# B&R Automation Studio project perfxxl (part 6)

#### seriell.c
```c
#ifdef _DEFAULT_INCLUDES
	#include <AsDefault.h>
#endif
/**
                             *******************
******************************* C SOURCE FILE *******************************
**                           *******************                           **
**                                                                         **
** project  : LS JET II                                                    **
** filename : SERIELL.C                                                    **
** version  : 1.12                                                         **
** date     : 15.06.2010                                                   **
**                                                                         **
*****************************************************************************
**                                                                         **
** Abstract                                                                **
** ========                                                                **
** Implementation of serial communication with Faulhaber motor units       **
** - cyclic polling of current position                                    **
** - send commands to a specific motors                                    **
** - request data from a specific motor                                    **
**                                                                         **
**                                                                         **
** Copyright (c) 2006, Krause-Biagosch GmbH                                **
** All rights reserved.                                                    **
**                                                                         **
*****************************************************************************
VERSION HISTORY:
----------------
Version     : 1.00
Date        : 05.09.2002
Revised by  : Herbert Aden
Description : Original version.

Version     : 1.10
Date        : 30.09.2002
Revised by  : Herbert Aden
Description : If a timeout occurs, the Position request is repeated up to 5 times

Version     : 1.11
Date        : 17.10.2006
Revised by  : Herbert Aden
Description : - Code review, style improvement
              - only number of received chars is copied from receive-buffer now
              - RequestData is now local to this module

Version     : 1.12
Date        : 15.06.2010
Revised by  : Herbert Aden
Description : - generate errormessages from FaultStatus (overtemp., current limiting,
                under- or overvoltage)

Version     : 1.13
Date        : 26.04.2011
Revised by  : Herbert Aden
Description : - errormessage delayed to make sure the faultmotor is correctly set
                before the message shows up (avoid error: Motor 0 blahblah)

TODO: Error handling, if system calls fail
*/
#define _SERIELL_C_SRC

/****************************************************************************/
/**                                                                        **/
/**                           INCLUDE FILES                                **/
/**                                                                        **/
/****************************************************************************/
#include <bur/plctypes.h>
#include <string.h>
#include <AsString.h>
#include <dvframe.h>
#include <standard.h>
#include <math.h>

#include "glob_var.h"
#include "sys_lib.h"
#include "motorfunc.h"

/****************************************************************************/
/**                                                                        **/
/**                       DEFINITIONS AND MACROS                           **/
/**                                                                        **/
/****************************************************************************/
#define BROADCAST 127	/* also in motorstop.c !! */
#define DATA_RECEIVED	0
#define STATUS_OK	0

/****************************************************************************/
/**                                                                        **/
/**                           GLOBAL VARIABLES                             **/
/**                                                                        **/
/****************************************************************************/
/*@-exportlocal@*/
/* stop lint from complainig, these are used in another task and therefore GLOBAL*/
_GLOBAL	RTCtime_typ		RTCtime;
_GLOBAL	USINT			MotorTemp[MAXMOTORS],MaxMotorTemp[MAXMOTORS];
_GLOBAL	STRING			MotorFaultStatus[MAXMOTORS][5];
_GLOBAL	DINT			MotorCurrent[MAXMOTORS],MaxMotorCurrent[MAXMOTORS];
/*@+exportlocal@*/

/****************************************************************************/
/**                                                                        **/
/**                      TASK-LOCAL VARIABLES                              **/
/**                                                                        **/
/****************************************************************************/
/* NONE */
_LOCAL	BOOL			GetMotorCurrent;			/* command to get the motor current*/
_LOCAL	UINT            FaultMotor;                 /* for Alarmmessage */
_LOCAL	DINT BufLng;
_LOCAL	STRING DebugBuf[64];

/****************************************************************************/
/**                                                                        **/
/**                    MODULE-LOCAL VARIABLES                              **/
/**                                                                        **/
/****************************************************************************/
static	UINT 			Counter;
static	UINT 			SendWaitCounter;
static	UINT			GetTempStep;
static	UINT			GetTempMotor;
static	USINT			lastSecond;
static	UINT			SecondCounter;
static	BOOL			xopenOK;					/* Opening the interface was successful*/
static	INT 			i;
static 	USINT 			RequestData[READDATALENGTH]; 			/* array for requested Data */
static 	char 			StringDevice[30], StringMode[30]; 		/* initialize strings for FRM_xopen */
static 	UINT 			timeout;
static	UINT 			Motor;						/* index variable for polling loop*/
static	BOOL 			StopPolling;				/* stop polling loop to send a command*/
static	UINT 			PollingStep;
static	UINT 			RequestStep;
static 	UINT			ResendCounter;
static	BOOL			GetMotorCurrentMem;			/* to detect changing of command*/
static	INT				Error;						/* Error Number for debugging*/
static	INT				ReceivedChar;
static	char		    tmp[20];
static	FRM_xopen_typ 	FrameXOpenStruct;
static	FRM_close_typ 	FrameCloseStruct;
static	XOPENCONFIG 	XOpenConfigStruct;
static	FRM_gbuf_typ 	FrameGetBufferStruct;
static	FRM_rbuf_typ 	FrameReleaseBufferStruct;
static	FRM_robuf_typ 	FrameReleaseOutputBufferStruct;
static	FRM_write_typ 	FrameWriteStruct;
static 	FRM_read_typ 	FrameReadStruct;
static  TON_10ms_typ    Alarm36Delay,Alarm37Delay,Alarm38Delay,Alarm39Delay;

/****************************************************************************/
/**                                                                        **/
/**                          LOCAL FUNCTIONS                               **/
/**                                                                        **/
/****************************************************************************/

/**
 * Return the next motor-number in the row, skipping those that are not
 * used in differently equipped machines
 *
 * Input Parameter: Current motor-number
 *
 * Returns        : Next motor-number
 *
 */
static UINT	NextMotor(UINT lMotor)
{
	lMotor++;
	if(lMotor == FEEDER_HORIZONTAL && !GlobalParameter.FlexibleFeeder)
		lMotor++;
	if(lMotor == ADJUSTER)
		lMotor++;
	if(lMotor == SHUTTLE)
		lMotor++;
	if(lMotor == DELOADER_TURN && GlobalParameter.DeloaderTurnStation != DELOADER_AND_TURNSTATION)
		lMotor++;
	if(lMotor == DELOADER_HORIZONTAL && GlobalParameter.DeloaderTurnStation == NO_DELOADER)
		lMotor++;

	if(lMotor > MotorsConnected)
		lMotor = 1;

	return lMotor;
}

/**
 * Auxiliary function to handle timeout while reading from serial interface
 *
 * Input Parameter: ----
 *
 * Returns        : ----
 *
 */
static void HandleTimeout(int returnstep)
{
	Error = 5; 						/* set error level for FRM_read */
	timeout++;
	if (timeout == 60) /* 60*cyclic (->300ms) time no answer */
	{
		if(ResendCounter == 5) /*5 times tried? -> error*/
		{
			ResendCounter = 0;
			Motors[Motor].Error = TRUE;
			Motors[Motor].Moving = FALSE;
			Motors[Motor].MovingPlus = FALSE;
			Motors[Motor].MovingMinus = FALSE;
			Motors[Motor].ReferenceOk = FALSE;
			Motor = NextMotor(Motor);
			if(Motor == 1)
				Counter++;

			PollingStep = 0;
		}
		else
		{
			ResendCounter++;
			PollingStep = /*1*/returnstep;
		}
	}
}

/**
 * Auxiliary function to handle error while writing to serial interface
 *
 * Input Parameter: ----
 *
 * Returns        : ----
 *
 */
static void HandleWriteError(void)
{
	/* initialize release output buffer structure */
	FrameReleaseOutputBufferStruct.buffer = FrameGetBufferStruct.buffer;
	FrameReleaseOutputBufferStruct.buflng = FrameGetBufferStruct.buflng;
	FRM_robuf(&FrameReleaseOutputBufferStruct); 	/* release output buffer */

	Error = 3; 					/* set error level for FRM_write */

	if (FrameReleaseOutputBufferStruct.status != 0) 		/* check status */
	{
		Error = 4; 				/* set error level for FRM_robuf */
	}
}

/**
 * Auxiliary function to handle error while writing to serial interface
 *
 * Input Parameter: ----
 *
 * Returns        : ----
 *
 * TODO: Error handling
 */
static void ReleaseBuffer(void)
{
	/* initialize release buffer structure */
	FrameReleaseBufferStruct.buffer = FrameReadStruct.buffer;	/* get adress of read buffer */
	FrameReleaseBufferStruct.buflng = FrameReadStruct.buflng; 	/* get length of read buffer */

	FRM_rbuf(&FrameReleaseBufferStruct); 			/* release read buffer */

	if (FrameReleaseBufferStruct.status != 0) 				/* check status */
	{
		Error = 6; 					/* set error level for FRM_rbuf */
	}
}

/****************************************************************************/
/** Init function, executed once at startup                                **/
/****************************************************************************/
_INIT void InitProgram(void)
{
	Alarm36Delay.IN = FALSE;
	Alarm37Delay.IN = FALSE;
	Alarm38Delay.IN = FALSE;
	Alarm39Delay.IN = FALSE;
	GetMotorCurrent = FALSE;
	GetMotorCurrentMem = FALSE;
	GetTempMotor = 1;
	lastSecond = US(0);
	SecondCounter = 0;
	for(i=0;i<MAXMOTORS;i++)
	{
		MotorTemp[i] = US(0);
		MaxMotorTemp[i] = US(0);
		MotorCurrent[i] = L(0);
		MaxMotorCurrent[i] = L(0);
	}

	/* initialize start values */
	Motor = 1;
/* Motor Nummern sind 1,2,3,6,9
 * um die Zuordnung zwischen Adr. und Fkt. wie beim Jet2 zu haben
 */
	MotorsConnected = 10;
	SendWaitCounter=0;
	Counter = 0;
	StopPolling = FALSE;
	ResendCounter = 0;
	xopenOK = 0;
	strcpy(&StringDevice[0], "IF1"); 							/* interface #1 */
	strcpy(&StringMode[0], "/BD=19200 /PA=N /DB=8 /SB=1"); 		/* RS232 interface, 19200 BAUD, no parity, 8 data bits, 1 stop bit */

	/* initialize config structure */
	XOpenConfigStruct.idle = 6;                           	/* in Zeichenlängen*/
	XOpenConfigStruct.delimc = 1;
	XOpenConfigStruct.delim[0] = (unsigned char)10;				/* LF */
	XOpenConfigStruct.delim[1] = (unsigned char)13;				/* CR */
	XOpenConfigStruct.tx_cnt = 6;
	XOpenConfigStruct.rx_cnt = 6;
	XOpenConfigStruct.tx_len = 64;
	XOpenConfigStruct.rx_len = 64;
	XOpenConfigStruct.argc = 0;
	XOpenConfigStruct.argv = 0;

	/* initialize open structure */
	FrameXOpenStruct.enable = TRUE;
	FrameXOpenStruct.device = (UDINT) StringDevice;
	FrameXOpenStruct.mode = (UDINT) StringMode;
	FrameXOpenStruct.config = (UDINT) &XOpenConfigStruct;

	FRM_xopen(&FrameXOpenStruct); 						/* open an interface */

	if (FrameXOpenStruct.status == 0) 					/* check status */
	{
		xopenOK = TRUE;									/* set error level for FRM_xopen */

		/* initialize get buffer structure */
		FrameGetBufferStruct.enable = TRUE;
		FrameGetBufferStruct.ident = FrameXOpenStruct.ident;				/* get ident */

		/* initialize write structure */
		FrameWriteStruct.enable = TRUE;
		FrameWriteStruct.ident  = FrameXOpenStruct.ident;					/* get ident */

		/* initialize release output buffer structure */
		FrameReleaseOutputBufferStruct.enable = TRUE;
		FrameReleaseOutputBufferStruct.ident = FrameXOpenStruct.ident;		/* get ident */

		/* initialize read structure */
		FrameReadStruct.enable = TRUE;
		FrameReadStruct.ident = FrameXOpenStruct.ident;						/* get ident */

		/* initialize release buffer structure */
		FrameReleaseBufferStruct.enable = TRUE;
		FrameReleaseBufferStruct.ident = FrameXOpenStruct.ident;			/* get ident */

		/* initialize close structure */
		FrameCloseStruct.enable = TRUE;
		FrameCloseStruct.ident = FrameXOpenStruct.ident;					/* get ident */
	}
	else
	{
		xopenOK = FALSE;
	}
}

/****************************************************************************/
/** Cyclic function                                                        **/
/****************************************************************************/
_CYCLIC void CyclicProgram(void)
{
/*HA 24.02.04 V1.76 reset MaxCurrent on activating measurement*/
	if ( GetMotorCurrent && !GetMotorCurrentMem )
		for(i=0;i<MAXMOTORS;i++)
			MaxMotorCurrent[i] = 0;
	GetMotorCurrentMem = GetMotorCurrent;

	if (xopenOK != FALSE)
	{
/******************************************************************/
/* Cyclic polling of current Positions */
/******************************************************************/
		switch (PollingStep)
		{
			case 0:
			{
				if(StopPolling) break;
				/*Safety: priority 0 doesn't make sense*/
				if(Motors[Motor].Parameter.Priority == US(0)) Motors[Motor].Parameter.Priority = US(1);

				if( (Counter % Motors[Motor].Parameter.Priority) == 0  )
				{
					PollingStep = 100;
				}
				else
				{
					Motor = NextMotor(Motor);
					if(Motor == 1)
						Counter++;
				}
				ResendCounter = 0;
				break;
			}

/* clear buffer from any unwanted msg */
			case 100:
			{
				/* initialize read structure */
				FRM_read(&FrameReadStruct); 						/* read data form interface */

				if (FrameReadStruct.status == DATA_RECEIVED) 					/* Data received */
				{
					ReleaseBuffer();
				}
				ResendCounter = 0;
				PollingStep = 1;
				break;
			}

/* 1st Step: send the POS command */
			case 1:
			{
				FRM_gbuf(&FrameGetBufferStruct); 				/* get send buffer */

				if (FrameGetBufferStruct.status == 0) 			/* check status */
				{
					size_t length = 4; /* length of "xPOS" */
					char *ptr = (char *)FrameGetBufferStruct.buffer;
				/*fill the buffer */
					(void) itoa(L(Motor),(UDINT) ptr);
					strcat(ptr,"POS\r\n");
					length = strlen(ptr);

					/* initialize write structure */
					FrameWriteStruct.buffer = FrameGetBufferStruct.buffer;
					FrameWriteStruct.buflng = length+1;
					FRM_write(&FrameWriteStruct); 				/* write data to interface */

					if (FrameWriteStruct.status != 0) 			/* check status */
					{
						HandleWriteError();
					}
				}
	/*TODO: Fehler auswerten wenn getBuffer fehlschlägt (8071)*/
				PollingStep++;
				timeout = 0;
				break;
			}
/* wait for the answer of Motor*/
			case 2:
			{
				/* initialize read structure */
				FRM_read(&FrameReadStruct); 						/* read data form interface */

				if (FrameReadStruct.status == DATA_RECEIVED) 					/* Data received */
				{
					BufLng = FrameReadStruct.buflng;
					strncpy(DebugBuf,((char *)FrameReadStruct.buffer),sizeof(DebugBuf));
					DebugBuf[BufLng] = '\0';
					if( (((char *)FrameReadStruct.buffer)[0] == '-')
					 || (   (((char *)FrameReadStruct.buffer)[0] >= '0')
					      &&(((char *)FrameReadStruct.buffer)[0] <= '9')
					    )
					  )
					{
						Motors[Motor].LastPosition = Motors[Motor].Position;
						Motors[Motor].Position = atoi( FrameReadStruct.buffer);
	/*@-realcompare@*/
						if(Motors[Motor].Parameter.IncrementsPerMm > 1.0)
							Motors[Motor].Position_mm = Motors[Motor].Position / Motors[Motor].Parameter.IncrementsPerMm;
	/*@+realcompare@*/

						if (Motor == ADJUSTER ||  Motor == CONVEYORBELT)
						{
							AbsMotorPos[Motor] = Motors[Motor].Position;
							AbsMotorPosMm[Motor] = Motors[Motor].Position_mm;
						}
						else
						{
							AbsMotorPos[Motor] = abs(Motors[Motor].Position);
							AbsMotorPosMm[Motor] = fabs(Motors[Motor].Position_mm);
						}

						if( labs(Motors[Motor].Position) > labs(Motors[Motor].LastPosition) )
						{
							Motors[Motor].MovingPlus = TRUE;
							Motors[Motor].MovingMinus = FALSE;
						}
						else
						{
							Motors[Motor].MovingPlus = FALSE;
							Motors[Motor].MovingMinus = TRUE;
						}

						if( labs(Motors[Motor].LastPosition - Motors[Motor].Position) > 100)
							Motors[Motor].Moving = TRUE;
						else
						{
							Motors[Motor].Moving = FALSE;
							Motors[Motor].MovingPlus = FALSE;
							Motors[Motor].MovingMinus = FALSE;
						}

						Motors[Motor].Error = FALSE;
					}
					ReleaseBuffer();
					if ( GetMotorCurrent )
					{
						PollingStep++;
						break;
					}
					else
					{
						Motor = NextMotor(Motor);
						if(Motor == 1)
							Counter++;

						PollingStep = 0;
						ResendCounter = 0;
						break;
					}
				}
				else	/* No data received or any error*/
				{
					HandleTimeout(1);
				}
				break;
			}
/* send the "get current" command*/
			case 3:
			{
					FRM_gbuf(&FrameGetBufferStruct); 				/* get send buffer */

					if (FrameGetBufferStruct.status == 0) 			/* check status */
					{
						size_t length = 4;
						char *ptr = (char *)FrameGetBufferStruct.buffer;
				/*fill the buffer */
						(void) itoa(L(Motor),(UDINT) ptr);
						strcat(ptr,"GRC\r\n"); /*actual current (Get Real Current)*/
						length = strlen(ptr);

					/* initialize write structure */
						FrameWriteStruct.buffer = FrameGetBufferStruct.buffer;		/* get adress of send buffer */
						FrameWriteStruct.buflng = length+1;

						FRM_write(&FrameWriteStruct); 				/* write data to interface */

						if (FrameWriteStruct.status != 0) 			/* check status */
						{
							HandleWriteError();
						}
					}
	/*TODO: Fehler auswerten wenn getBuffer fehlschlägt (8071)*/
					PollingStep++;
					timeout = 0;
					break;
			}

/* wait for the answer of Motor on GRC*/
			case 4:
			{
				/* initialize read structure */
				FRM_read(&FrameReadStruct); 						/* read data form interface */

				if (FrameReadStruct.status == DATA_RECEIVED) 					/* Data received */
				{
					if( (((char *)FrameReadStruct.buffer)[0] == '-')
					 || (   (((char *)FrameReadStruct.buffer)[0] >= '0')
					      &&(((char *)FrameReadStruct.buffer)[0] <= '9')
					    )
					  )
					{
						MotorCurrent[Motor] = atoi( FrameReadStruct.buffer);
						if ( MotorCurrent[Motor] > MaxMotorCurrent[Motor] )
							MaxMotorCurrent[Motor] = MotorCurrent[Motor];
					}
					ReleaseBuffer();

					Motor = NextMotor(Motor);
					if(Motor == 1)
						Counter++;

					PollingStep = 0;
					ResendCounter = 0;
					break;
				}
				else	/* No data received or any error*/
				{
					HandleTimeout(3);
				}
				break;
			}

		} /*switch*/

/******************************************************************/
/* requesting of Parameter */
/******************************************************************/
		switch (RequestStep)
		{
			case 0:
			{
				if(SerialCmd.Send == FALSE) break; /*wait for send command*/

				StopPolling = TRUE;
				if(PollingStep == 0)	/*wait for polling to stop*/
					RequestStep++;
				break;
			}
/* 1st Step: send the command */
			case 1:
			{
				FRM_gbuf(&FrameGetBufferStruct); 				/* get send buffer */

				if (FrameGetBufferStruct.status == STATUS_OK)
				{
					size_t length=0; /* length */
					char *ptr = (char *)FrameGetBufferStruct.buffer;
				/*fill the buffer */
					if( SerialCmd.SendMotor != BROADCAST )  /*no BROADCAST, so the address must be first*/
					{
						(void)itoa(L(SerialCmd.SendMotor),(UDINT) ptr);
						strcat(ptr,(char *) SerialCmd.CmdString);
					}
					else
						strcpy(ptr,(char *) SerialCmd.CmdString);

/* build the final commandstring from given parameters*/
					if (SerialCmd.UseParameter)
					{
						if (SerialCmd.UseRefDirection)
						{
				/*
				 * for absolute positioning:
				 * if Reference direction positive then the way to move is in negative direction
				 * therefore labs(SerialCmd.Parameter)
				*/
							if (STREQ(SerialCmd.CmdString,CMD_ABSOLUTE_POS))
							{
								if( (SerialCmd.SendMotor == CONVEYORBELT) || (SerialCmd.SendMotor == ADJUSTER) )
								{
							/*
							 * special case: the belt drives are able to move in a position below 0
							 * so this is allowed here in that special case
							*/
									(void)itoa(SerialCmd.Parameter,(UDINT) &tmp[0]);
								}
								else
								{
									if (Motors[SerialCmd.SendMotor].Parameter.ReferenceDirectionNegative == FALSE)
										strcat(ptr,"-");
									(void)itoa(labs(SerialCmd.Parameter),(UDINT) &tmp[0]);
								}
							}
							else
				/*
				 * for relative positioning:
				 * moving towards reference pos. must be given as negative values
				 * UseRefDirection must be TRUE
				 * the same applies for speed setting (V-command)
				*/

							if ( (STREQ(SerialCmd.CmdString,CMD_RELATIVE_POS))
								||
								(STREQ(SerialCmd.CmdString,CMD_MOVE_AT)))
							{
								if(Motors[SerialCmd.SendMotor].Parameter.ReferenceDirectionNegative)
								{
									if (SerialCmd.Parameter < 0L)
										strcat(ptr,"-");
								}
								else
								{
									if (SerialCmd.Parameter > 0L)
										strcat(ptr,"-");
								}
								(void)itoa(labs(SerialCmd.Parameter),(UDINT) &tmp[0]);
							}
						}
						else /* don't use RefDirection: take Parameter just as it's given */
							(void)itoa(SerialCmd.Parameter,(UDINT) &tmp[0]);

						strcat(ptr,tmp);
					}
					strcat(ptr,"\r\n");
					length = strlen(ptr);

					/* initialize write structure */
					FrameWriteStruct.buffer = FrameGetBufferStruct.buffer;	/* get adress of send buffer */
					FrameWriteStruct.buflng = length+1; 					/* set length of send buffer */

					FRM_write(&FrameWriteStruct); 				/* write data to interface */

					if (FrameWriteStruct.status != 0) 			/* check status */
					{
						HandleWriteError();
					}
				}
				RequestStep++;
				timeout = 0;
				break;
			}
/* wait for the answer of Motor*/
			case 2:
			{
				/* no request: go on*/
				if(SerialCmd.Request == FALSE)
				{
					SendWaitCounter++;
					if(SendWaitCounter > 6)
					{
						SendWaitCounter=0;
						SerialCmd.Request = FALSE;
						SerialCmd.Send = FALSE;
						StopPolling = FALSE;
						RequestStep = 0;
					}
/* HA 13.02.04 V1.76 no request (command only): leave the code immediately */
					break;
				}
/* otherwise go ahead waiting for answer*/

				/* initialize read structure */
				FRM_read(&FrameReadStruct); 						/* read data form interface */

				if (FrameReadStruct.status == DATA_RECEIVED) 					/* Data received */
				{
					ReceivedChar = (INT) FrameReadStruct.buflng;
					memcpy(RequestData, (USINT*)FrameReadStruct.buffer, (size_t)ReceivedChar); /* copy read data into array */
					Motors[SendMotor].Error = FALSE;

					ReleaseBuffer();

					RequestStep = 0;
					SerialCmd.Request = FALSE;
					SerialCmd.Send = FALSE;
					StopPolling = FALSE;
				}
				else	/* No data received or any error*/
				{
					ReceivedChar = 0;
					Error = 5; 						/* set error level for FRM_read */
					timeout++;
					if (timeout == 60) /* 60*cyclic time no answer */
					{
						RequestStep = 0;
						SerialCmd.Request = FALSE;
						SerialCmd.Send = FALSE;
						StopPolling = FALSE;
						Motors[SerialCmd.SendMotor].Error = TRUE;
						Motors[SerialCmd.SendMotor].Moving = FALSE;
						Motors[SerialCmd.SendMotor].MovingPlus = FALSE;
						Motors[SerialCmd.SendMotor].MovingMinus = FALSE;
					}
				}
				break;
			}
		} /*switch*/

	} /*if (xopenOK == 1)*/

/******************************************************************************************************/
/******************************************************************************************************/
/******************************************************************************************************/
/* Alarm 36 bis 39 5s verzögern, damit der Faultmotor auch sicher eingetragen wurde */
	Alarm36Delay.PT = 500;
	TON_10ms(&Alarm36Delay);
	AlarmBitField[36] = Alarm36Delay.Q;

	Alarm37Delay.PT = 500;
	TON_10ms(&Alarm37Delay);
	AlarmBitField[37] = Alarm37Delay.Q;

	Alarm38Delay.PT = 500;
	TON_10ms(&Alarm38Delay);
	AlarmBitField[38] = Alarm38Delay.Q;

	Alarm39Delay.PT = 500;
	TON_10ms(&Alarm39Delay);
	AlarmBitField[39] = Alarm39Delay.Q;

	switch (GetTempStep)
	{
/* get Temperature every 5 seconds*/
		case 0:
		{
			int CurrentMotor=1,j=0;
/*Fehlermedlungen zurücksetzen, wenn alle Motoren keinen Fehler mehr melden */
			while(CurrentMotor <= MotorsConnected)
			{
				if(CurrentMotor == FEEDER_HORIZONTAL && !GlobalParameter.FlexibleFeeder)
					CurrentMotor++;
				if(CurrentMotor == ADJUSTER)
					CurrentMotor++;
				if(CurrentMotor == SHUTTLE)
					CurrentMotor++;

				if(   (CurrentMotor == DELOADER_TURN)
				   && (GlobalParameter.DeloaderTurnStation != DELOADER_AND_TURNSTATION) )
					CurrentMotor++;

				if(   (CurrentMotor == DELOADER_HORIZONTAL)
				   && (GlobalParameter.DeloaderTurnStation == NO_DELOADER) )
					CurrentMotor++;

				if( !STREQ(MotorFaultStatus[CurrentMotor],"0000"))
					j++;

				CurrentMotor++;
			}

			if( j == 0 )
			{
				Alarm36Delay.IN = FALSE;
				Alarm37Delay.IN = FALSE;
				Alarm38Delay.IN = FALSE;
				Alarm39Delay.IN = FALSE;
				AlarmBitField[36] = FALSE;
				AlarmBitField[37] = FALSE;
				AlarmBitField[38] = FALSE;
				AlarmBitField[39] = FALSE;
			}

			if( RTCtime.second != lastSecond)
			{
				if(SecondCounter >= 5 )
				{
					GetTempStep = 1;
					SecondCounter = 0;
				}
				else
					SecondCounter++;
				lastSecond = RTCtime.second;
				break;
			}
			break;
		}
		case 1:
		{
			if(Motors[GetTempMotor].Error)
			{
				GetTempMotor = NextMotor(GetTempMotor);
				GetTempStep = 0;
				break;
			}

			if( SerialCmd.Send == FALSE )
			{
				if( RequestMotorData(GetTempMotor,CMD_GETTEMP) )
					GetTempStep = 5;
				break;
			}
			break;
		}

		case 5:
		{
			if(SerialCmd.Request == FALSE)
			{
				if(  ReceivedChar != 0
			     && !Motors[SerialCmd.SendMotor].Error )
			    {
					MotorTemp[GetTempMotor] = US(atoi( (UDINT) &RequestData[0]));
					if ( MotorTemp[GetTempMotor] > MaxMotorTemp[GetTempMotor] )
					{
						MaxMotorTemp[GetTempMotor] = MotorTemp[GetTempMotor];
					}
				}
				GetTempStep = 10;
			}
			break;
		}
		case 10:
		{
			if ( RequestMotorData(GetTempMotor,CMD_GETFAULTSTAT) )
				GetTempStep = 15;

			break;
		}
		case 15:
		{
			if( SerialCmd.Request == FALSE )
			{
				if(  ReceivedChar != 0
			     && !Motors[SerialCmd.SendMotor].Error )
			    {
					memcpy(&MotorFaultStatus[GetTempMotor][0],&RequestData[0],4);
					MotorFaultStatus[GetTempMotor][4] = 0;
					if(MotorFaultStatus[GetTempMotor][0] == '1')
					{/* Übertemp. */
						Alarm36Delay.IN = TRUE;
						FaultMotor = GetTempMotor;
					}
					if(   Motors[GetTempMotor].ReferenceOk
					  && (MotorFaultStatus[GetTempMotor][1] == '1') )
					{/* Überstrom */
						Alarm37Delay.IN = TRUE;
						FaultMotor = GetTempMotor;
					}
					if(MotorFaultStatus[GetTempMotor][2] == '1')
					{/* Unterspannung */
						Alarm38Delay.IN = TRUE;
						FaultMotor = GetTempMotor;
					}
					if(MotorFaultStatus[GetTempMotor][3] == '1')
					{/* Überspannung */
						Alarm39Delay.IN = TRUE;
						FaultMotor = GetTempMotor;
					}
				}

				GetTempMotor = NextMotor(GetTempMotor);
				GetTempStep = 0;
			}
			break;
		}
	}

}

/****************************************************************************/
/**                                                                        **/
/**                                 EOF                                    **/
/**                                                                        **/
/****************************************************************************/
```

- glob_var.h (reference to Logical/GlobalIncludes/glob_var.h)

- motorfunc.h (reference to Logical/GlobalIncludes/motorfunc.h)

#### motorfunc.c
```c
#ifdef _DEFAULT_INCLUDES
	#include <AsDefault.h>
#endif
/*
                             *******************
******************************* C SOURCE FILE *******************************
**                           *******************                           **
**                                                                         **
** project  : LS JET II                                                    **
** filename : MOTORFUNC.C                                                  **
** version  : 1.02                                                         **
** date     : 07.11.2007                                                   **
**                                                                         **
*****************************************************************************
** Abstract                                                                **
** ========                                                                **
** Implementation of motor control functions (sending commands and         **
** check for positions)                                                    **
**                                                                         **
** Copyright (c) 2007, Krause-Biagosch GmbH                                **
** All rights reserved.                                                    **
**                                                                         **
*****************************************************************************
VERSION HISTORY:
----------------
Version     : 1.00
Date        : 20.10.2006
Revised by  : Herbert Aden
Description : Original version.

Version     : 1.01
Date        : 12.10.2007
Revised by  : Herbert Aden
Description : - a variable for holding the current step in function MoveToAbsPosition
                must now be provided by the caller (a pointer to that var of course!)
              - in Fct. IsPositionOK the check for being in a certain position window
                failed, if that window was 0, i.e. if an exact position is to be found
                the expression "currpos - checkpos < deviation" results in false, so it
                was changed to "currpos - checkpos <= deviation" so that if
                currpos==checkpos the result is still true for deviaition==0

Version     : 1.02
Date        : 07.11.2007
Revised by  : Herbert Aden
Description : - bugfix: in RequestMotorData the var SerialCmd.Request was set TRUE
                unconditionally. Caused sporadic Errormessages for serial comm.

*/
#define _MOTORFUNC_C_SRC

/****************************************************************************/
/**                                                                        **/
/**                           INCLUDE FILES                                **/
/**                                                                        **/
/****************************************************************************/
#include "glob_var.h"
#include "AsBrStr.h"
#include <stdlib.h>
#include <string.h>

#include "motorfunc.h"

/****************************************************************************/
/**                                                                        **/
/**                       DEFINITIONS AND MACROS                           **/
/**                                                                        **/
/****************************************************************************/
/* NONE */

/****************************************************************************/
/**                                                                        **/
/**                      EXPORTED VARIABLES                                **/
/**                                                                        **/
/****************************************************************************/
/*@checked@*/
_GLOBAL   SerialCmd_Typ       SerialCmd;

/****************************************************************************/
/**                                                                        **/
/**                           GLOBAL VARIABLES                             **/
/**                                                                        **/
/****************************************************************************/
static  BOOL                  Send1Ready = 0;

/****************************************************************************/
/**                                                                        **/
/**                          EXPORTED FUNCTIONS                            **/
/**                                                                        **/
/****************************************************************************/

/****************************************************************************/
/** Send commands to a motor                                                */
/****************************************************************************/
BOOL	SendMotorCmd(const INT pMotor,const char *CmdStr,const BOOL UseValue,const DINT Value)
{
	if(SerialCmd.Send == FALSE) /*wait, till no other sending active*/
	{
		strcpy(SerialCmd.CmdString,CmdStr);
		SerialCmd.UseParameter = UseValue;
		SerialCmd.Parameter = Value;
		if (   (STREQ(CmdStr,CMD_ABSOLUTE_POS))
			|| (STREQ(CmdStr,CMD_RELATIVE_POS))
			|| (STREQ(CmdStr,CMD_MOVE_AT))
		  ) /*bei LA oder LR oder V Refdir verwenden, sonst nicht*/
			SerialCmd.UseRefDirection = TRUE;
		else
			SerialCmd.UseRefDirection = FALSE;

		SerialCmd.SendMotor = pMotor;
		SerialCmd.Send = TRUE;
		return TRUE;
	}
	else
		return FALSE;
}

/****************************************************************************/
/** Request data from a motor                                                */
/****************************************************************************/
BOOL	RequestMotorData(const INT pMotor,const char *CmdString)
{
	if( SerialCmd.Send == TRUE )
		return FALSE;
	else
	{
		SerialCmd.Request = TRUE;
		return SendMotorCmd(pMotor,CmdString,FALSE,0);
	}
}

/****************************************************************************/
/** Check, if a motor is in a certain position window                       */
/****************************************************************************/
BOOL	isPositionOk(const INT Motor,const DINT Pos,const DINT Deviation)
{
	DINT tmp;
	if (labs(Deviation) > 0 )
		tmp = labs(Deviation);
	else	/* if Dev is 0, then use deviation defined in motorparam*/
		tmp = labs(Motors[Motor].Parameter.PositionWindow);

	if( labs( labs(Motors[Motor].Position) - labs(Pos) ) <= tmp )
		return TRUE;
	else
		return FALSE;
}

/****************************************************************************/
/** Check, if a motor is below a certain position                           */
/****************************************************************************/
BOOL	isPositionLowerThan(const INT Motor,DINT Pos)
{
	if( labs(Motors[Motor].Position) < (labs(Pos) ) )
		return TRUE;
	else
		return FALSE;
}

/****************************************************************************/
/** Check, if a motor is above a certain position                           */
/****************************************************************************/
BOOL	isPositionHigherThan(const INT Motor,DINT Pos)
{
	if( labs(Motors[Motor].Position) > (labs(Pos) ) )
		return TRUE;
	else
		return FALSE;
}

/****************************************************************************/
/* send commands to paper remove vertical */
/****************************************************************************/
BOOL	PapRemVerticalCmd(BOOL Config,char *CmdString,BOOL UseValue,DINT Value)
{
	if(Config == LEFT)
		return SendMotorCmd(PAPERREMOVE_VERTICAL, CmdString, UseValue, Value);
	else
	if(Config == RIGHT)
		return SendMotorCmd(PAPERREMOVE_VERTICAL2, CmdString, UseValue, Value);
	else
	if ( Send1Ready == FALSE )
	{
		if( SendMotorCmd(PAPERREMOVE_VERTICAL, CmdString, UseValue, Value) )
			Send1Ready = TRUE;

		return FALSE;
	}
	else
	{
		if( SendMotorCmd(PAPERREMOVE_VERTICAL2, CmdString, UseValue, Value) )
		{
			Send1Ready = FALSE;
			return TRUE;
		}
		return FALSE;
	}
}

/****************************************************************************/
/* Check position of paper remove vertical */
/****************************************************************************/
BOOL	isPapRemVerticalOk(BOOL Config,DINT Pos,UDINT MaxDeviation)
{
	if(Config == LEFT)
		return isPositionOk(PAPERREMOVE_VERTICAL, Pos, MaxDeviation);
	else
	if(Config == RIGHT)
		return isPositionOk(PAPERREMOVE_VERTICAL2, Pos, MaxDeviation);
	else
	if ( isPositionOk(PAPERREMOVE_VERTICAL, Pos, MaxDeviation) )
	{
		if ( isPositionOk(PAPERREMOVE_VERTICAL2, Pos, MaxDeviation) )
			return TRUE;
		else
			return FALSE;
	}
	else
		return FALSE;
}

/****************************************************************************/
/* move motor to an absolute position and wait for motion to start */
/****************************************************************************/
BOOL  MoveToAbsPosition(INT pMotor, DINT Pos, DINT Speed, USINT *pStep)
{
	int step = *pStep;

	BOOL retval = FALSE;

	if (pMotor == 0 && Pos == 0L && Speed == 0L)
	{
		step = 0;
		*pStep = 0;
		return FALSE;
	}

	switch (step)
	{
		case 0:
		{
/* send target position */
			if( SendMotorCmd(pMotor,CMD_ABSOLUTE_POS,TRUE,Pos) )
			{
				if ( Speed == DONT_SEND_SPEED )
					step = 20;
				else
					step = 10;
			}
			retval = FALSE;
			break;
		}
/* set speed */
		case 10:
		{
			if( SendMotorCmd(pMotor,CMD_SPEED,TRUE,Speed) )
			{
				step = 20;
			}
			retval = FALSE;
			break;
		}
		case 20:
		{
/* start motion */
			if( SendMotorCmd(pMotor,CMD_START_MOTION,FALSE,0L) )
			{
				step = 30;
			}
			retval = FALSE;
			break;
		}
		case 30:
		{
/* Wait til motion begins or Motor is in position (might be already there!)*/
			if( Motors[pMotor].Moving
			    ||
			    isPositionOk(pMotor,Pos,0) )
			{
				step = 0;
				retval = TRUE;
			}
			break;
		}
	}
	*pStep = step;
	return retval;
}

/****************************************************************************/
/* move motor to an relative position without waiting for motion to start */
/****************************************************************************/
BOOL  MoveToRelPosition(INT pMotor, DINT Pos, DINT Speed, USINT *pStep)
{
	int step = *pStep;

	BOOL retval = FALSE;

	if (pMotor == 0 && Pos == 0L && Speed == 0L)
	{
		step = 0;
		*pStep = 0;
		return FALSE;
	}

	switch (step)
	{
		case 0:
		{
/* send target position */
			if( SendMotorCmd(pMotor,CMD_RELATIVE_POS,TRUE,Pos) )
			{
				if ( Speed == DONT_SEND_SPEED )
					step = 20;
				else
					step = 10;
			}
			retval = FALSE;
			break;
		}
/* set speed */
		case 10:
		{
			if( SendMotorCmd(pMotor,CMD_SPEED,TRUE,Speed) )
			{
				step = 20;
			}
			retval = FALSE;
			break;
		}
		case 20:
		{
/* start motion */
			if( SendMotorCmd(pMotor,CMD_START_MOTION,FALSE,0L) )
			{
				step = 30;
			}
			retval = FALSE;
			break;
		}
		case 30:
		{
			step = 0;
			retval = TRUE;
			break;
		}
	}
	*pStep = step;
	return retval;
}

/****************************************************************************/
/**                                                                        **/
/**                          LOCAL FUNCTIONS                               **/
/**                                                                        **/
/****************************************************************************/
/* NONE */

/****************************************************************************/
/**                                                                        **/
/**                                 EOF                                    **/
/**                                                                        **/
/****************************************************************************/
```

### Package Logical/Exposer/Ablauf - Funktionsabläufe

### Program Logical/Exposer/Ablauf/trolley (ANSIC, version 1.31.0) - Funktionen für Plattenwagen

#### trolley.c
```c
#ifdef _DEFAULT_INCLUDES
	#include <AsDefault.h>
#endif
/****************************************************************************/
/*	Plattenwagen Hauptprogramm */
/*																			*/
/*																			*/
/*	Versionsgeschichte:														*/
/*  Version		Datum		Änderung								von		*/
/*	1.0			10.09.02	erste Implementation					HA		*/
/*	1.31			02.04.03	Fehlerhandling:kein Pano Adapter			HA		*/
/*																			*/
/*																			*/
/****************************************************************************/

#include "glob_var.h"
#include "in_out.h"

_LOCAL	UINT	OpenTrolleyStep;
_LOCAL	USINT	CloseTrolleyStep;

_GLOBAL	BOOL	CloseTrolleyStart;
_GLOBAL	BOOL	OpenTrolleyStart;
_GLOBAL	BOOL	ReferenceStart,DontCloseTrolley;

_LOCAL TON_10ms_typ CloseTrolleyTimer;
_LOCAL TON_10ms_typ OpenTrolleyTimer;
_LOCAL F_TRIGtyp F_TRIG02;

extern void OpenTrolley(void);
extern void CloseTrolley(void);

extern void Test(void);

/****************************************************************************/
/* INIT Teil*/
/****************************************************************************/
_INIT void init(void)
{
	OpenTrolleyStep		= 0;
	OpenTrolleyStart	= 0;
	OpenTrolleyTimer.IN	= 0;
	OpenTrolleyTimer.PT	= 10; /*just to have any value in there...*/

	CloseTrolleyStep		= 0;
	CloseTrolleyStart		= 0;
	CloseTrolleyTimer.IN	= 0;
	CloseTrolleyTimer.PT	= 10; /*just to have any value in there...*/
	GlobalParameter.TrolleyLeft = 0;
	GlobalParameter.TrolleyRight = 0;
}

/****************************************************************************/
/* zyklischer Teil*/
/****************************************************************************/
_CYCLIC void cyclic(void)
{
	SequenceSteps[6] = (USINT) OpenTrolleyStep;
	SequenceSteps[7] = CloseTrolleyStep;

/*HA 26.06.03 V1.11 release cover lock, if machine is safe*/
	F_TRIG02.CLK =  AUTO
		|| START
		|| PaperRemoveStart
		|| PlateTakingStart
		|| AdjustStart
		|| DeloadStart
		|| ExposeStart
		|| CloseTrolleyStart
		|| OpenTrolleyStart
		|| PlateOnConveyorBelt.present
		|| PlateAtAdjustedPosition.present
		|| PlateAtDeloader.present
		|| ReferenceStart;

	F_TRIG(&F_TRIG02);
	if( F_TRIG02.Q )
	{
		Out_CoverLockOn = 0;
	}

/*error message if: trolley empty flag AND
Automatic Open/close and trolley is closed OR
no Automatic Open/close
*/
	if(TrolleyEmpty && ((GlobalParameter.AutomaticTrolleyOpenClose && !TrolleyOpen) || !GlobalParameter.AutomaticTrolleyOpenClose) )
	{
			if(PanoramaAdapter)
			{
				AlarmBitField[25]=1;
				AbfrageText1 = 37;
				AbfrageText2 = 40;
				AbfrageText3 = 0;
			}
			else
			{
				AlarmBitField[15]=1;
				AbfrageText1 = 17;
				AbfrageText2 = 18;
				AbfrageText3 = 19;
			}

			if(wBildAktuell != MESSAGEPIC )
				OrgBild = wBildAktuell;
			wBildNeu = MESSAGEPIC;
			AbfrageOK = 0;
			AbfrageCancel = 0;
			IgnoreButtons = 1;
			OK_CancelButtonInv = 1;
			OK_ButtonInv = 0;
			AbfrageIcon = CAUTION;
			TrolleyEmpty = 0;
	}

	OpenTrolley();
	CloseTrolley();
}
```

#### opentrolley.c
```c
#ifdef _DEFAULT_INCLUDES
	#include <AsDefault.h>
#endif
/****************************************************************************/
/*	Ablauf Plattenwagen öffnen */
/*																			*/
/*																			*/
/*	Versionsgeschichte:														*/
/*  Version		Datum		Änderung								von		*/
/*	1.00		10.09.02	erste Implementation					HA		*/
/*	1.10		16.09.02	Trolley offen/geschlossen jetzt mit		HA		*/
/*	1.20		02.01.03	vor oeffnen/schließen wird jetzt der	HA		*/
/*							Vertikalantrieb Referenz gefahren				*/
/*	1.30		06.01.03	Trolley erkennung implementiert			HA		*/
/*																			*/
/****************************************************************************/

#include "glob_var.h"
#include "in_out.h"
#include "asstring.h"
#include <string.h>
#include "Motorfunc.h"
#include "auxfunc.h"

#define PAPERREMOVEHORIZONTAL_MAXPOS (250000) /* Increments */
#define NO_TROLLEY (0)

_LOCAL	UINT	OpenTrolleyStep;
_GLOBAL	BOOL	OpenTrolleyStart;
_GLOBAL	BOOL	CloseTrolleyStart;
_LOCAL TON_10ms_typ OpenTrolleyTimer;

USINT			tmp[20];

_GLOBAL	BOOL	OpenTrolleyReady;

USINT	OpenCounter; /* for max 2 cycles (2 single trolleys)*/
_LOCAL CTUtyp TrolleyCodeCounter;
_LOCAL	UINT	DetectedTrolley,DetectionError,DetectCounter;
		DINT	StartPos,EndPos;
_GLOBAL	UINT	OrgBild,IgnoreButtons;

extern	STRING	NameTrolleyLeft[32],NameTrolleyRight[32];

static    BOOL                PaletteDetection;
static    BOOL                CheckForPalette;

void OpenTrolley(void)
{
	/* Motoren keine Referenz? -> Ende*/
	if( !Motors[PAPERREMOVE_VERTICAL].ReferenceOk
	||  !Motors[PAPERREMOVE_VERTICAL2].ReferenceOk
	)
		return;
	if( !Motors[PAPERREMOVE_HORIZONTAL].ReferenceOk ) return;
	if( !Motors[FEEDER_VERTICAL].ReferenceOk ) return;

	TON_10ms(&OpenTrolleyTimer);

	if (!OpenTrolleyStart) OpenTrolleyStep=0;

	switch (OpenTrolleyStep)
	{
		case 0:
		{
			DetectionError = 0;
			DetectCounter = 0;

/* wait for start command */
			if (!OpenTrolleyStart || PaperRemoveStart || CloseTrolleyStart) break;

/*enable conditions*/
/*check, if Feeder is out of collision area (should be the case here)*/
			if( abs(Motors[FEEDER_VERTICAL].Position) > abs(FeederParameter.VerticalPositions.EnablePaperRemove)+20 )
				break;

			OpenTrolleyTimer.IN = 0;

			OpenCounter = 1;

/*neuer Versuch: Alarme löschen */
			AlarmBitField[13] = 0;
			AlarmBitField[14] = 0;

/*NEW always do a reference of paperremove vert. at first */
			OpenTrolleyStep = 2;
			break;
		}

/*NEW paperremove vert reference at first*/
		case 2:
		{
			Motors[PAPERREMOVE_VERTICAL].StartRef = 1;
			Motors[PAPERREMOVE_VERTICAL].ReferenceOk = 0;
			Motors[PAPERREMOVE_VERTICAL2].StartRef = 1;
			Motors[PAPERREMOVE_VERTICAL2].ReferenceOk = 0;
			OpenTrolleyStep = 3;
			break;
		}
/*Wait for reference OK*/
/* then jump to 50 for trolley detection, if enabled, else go on with step 8*/
		case 3:
		{
			if( Motors[PAPERREMOVE_VERTICAL].ReferenceOk == 0
				|| Motors[PAPERREMOVE_VERTICAL2].ReferenceOk == 0
			)
				break;

			if( GlobalParameter.AutomaticTrolleyOpenClose)
				OpenTrolleyStep = 50;
			else
				OpenTrolleyStep = 8;
			break;
		}

		case 8:
		{
			if( (Out_PaperGripOn[LEFT] == 0)
			 && (Out_PaperGripOn[RIGHT] == 0)
			 && OpenTrolleyTimer.Q )
			{
				OpenTrolleyStep = 10;
				OpenTrolleyTimer.IN = 0;
				break;
			}

			Out_PaperGripOn[LEFT] = 0;
			Out_PaperGripOn[RIGHT] = 0;
			OpenTrolleyTimer.IN = 1;
			OpenTrolleyTimer.PT = PaperRemoveParameter.GripOffTime;
			break;
		}
		case 10:
		{

/*NEW*/
			if( (GlobalParameter.TrolleyLeft != 0) && OpenCounter == 1)
			{
			/* Palette: no opening -> ready, jump to final steps for moving back to parkpos */
				if(GlobalParameter.EnablePaletteLoading && Trolleys[GlobalParameter.TrolleyLeft].NoCover)
				{
					OpenTrolleyStep = 29;
					OpenTrolleyTimer.IN = FALSE;
					break;
				}
				PaperRemoveParameter.HorizontalPositions.TrolleyOpenRightStart = Trolleys[GlobalParameter.TrolleyLeft].OpenStart;
				PaperRemoveParameter.HorizontalPositions.TrolleyOpenRightStop = Trolleys[GlobalParameter.TrolleyLeft].OpenStop;
				PaperRemoveParameter.HorizontalPositions.TrolleyCloseRightStart = Trolleys[GlobalParameter.TrolleyLeft].CloseStart;
				PaperRemoveParameter.HorizontalPositions.TrolleyCloseRightStop = Trolleys[GlobalParameter.TrolleyLeft].CloseStop;
			}
			if( (GlobalParameter.TrolleyRight != 0 && OpenCounter == 2)
			||  (GlobalParameter.TrolleyLeft == 0 && GlobalParameter.TrolleyRight != 0 && OpenCounter == 1 ) )
			{
				PaperRemoveParameter.HorizontalPositions.TrolleyOpenRightStart = abs(Trolleys[GlobalParameter.TrolleyRight].OpenStart) + GlobalParameter.TrolleyRightOffset;
				PaperRemoveParameter.HorizontalPositions.TrolleyOpenRightStop = abs(Trolleys[GlobalParameter.TrolleyRight].OpenStop) + GlobalParameter.TrolleyRightOffset;
				PaperRemoveParameter.HorizontalPositions.TrolleyCloseRightStart = abs(Trolleys[GlobalParameter.TrolleyRight].CloseStart) + GlobalParameter.TrolleyRightOffset;
				PaperRemoveParameter.HorizontalPositions.TrolleyCloseRightStop = abs(Trolleys[GlobalParameter.TrolleyRight].CloseStop) + GlobalParameter.TrolleyRightOffset;
			}

/*check, if Feeder is out of collision area (should be the case here)*/
			if( abs(Motors[FEEDER_VERTICAL].Position) > abs(FeederParameter.VerticalPositions.EnablePaperRemove)+20 )
				break;

/*Move Paper remove horizontically to closed trolley pos*/
			if( SendMotorCmd(PAPERREMOVE_HORIZONTAL,"LA",TRUE,PaperRemoveParameter.HorizontalPositions.TrolleyOpenRightStart) )
				OpenTrolleyStep = 11;
			break;
		}
		case 11:
		{
/* Bewegung starten */
			if( SendMotorCmd(PAPERREMOVE_HORIZONTAL,"M",FALSE,0) )
				OpenTrolleyStep = 12;
			break;
		}
		case 12:
		{
/*Wait til Position is reached */
			if( isPositionOk(PAPERREMOVE_HORIZONTAL,PaperRemoveParameter.HorizontalPositions.TrolleyOpenRightStart,20) )
				OpenTrolleyStep = 14;

			break;
		}
		case 14:
		{
/* Paper remove down on trolley*/
			if( PapRemVerticalCmd(BOTH,CMD_SPEED,1,PaperRemoveParameter.TrolleyOpenDownSpeed) )
			{
				OpenTrolleyStep = 15;
			}
			break;
		}
		case 15:
		{
/* Paper remove down on trolley*/
			if( PapRemVerticalCmd(BOTH,CMD_ABSOLUTE_POS,TRUE,PaperRemoveParameter.VerticalPositions.OnTrolley) )
			{
				OpenTrolleyStep = 16;
			}
			break;
		}
		case 16:
		{
/* Bewegung starten */
			if( PapRemVerticalCmd(BOTH,CMD_START_MOTION,FALSE,0L) )
			{
				OpenTrolleyStep = 17;
			}
			break;
		}
		case 17:
		{
/*Wait for Pos*/
			if( isPapRemVerticalOk(BOTH,PaperRemoveParameter.VerticalPositions.OnTrolley,20) )
				OpenTrolleyStep = 19;
			break;
		}
		case 19:
		{
/*Move Paper remove horizontically to open trolley pos*/
			if( SendMotorCmd(PAPERREMOVE_HORIZONTAL,CMD_ABSOLUTE_POS,TRUE,PaperRemoveParameter.HorizontalPositions.TrolleyOpenRightStop) )
				OpenTrolleyStep = 20;
			break;
		}
		case 20:
		{
/*set speed */
			if( SendMotorCmd(PAPERREMOVE_HORIZONTAL,CMD_SPEED,TRUE,PaperRemoveParameter.TrolleyOpenCloseSpeed) )
				OpenTrolleyStep = 21;
			break;
		}
		case 21:
		{
/* Bewegung starten */
			if( SendMotorCmd(PAPERREMOVE_HORIZONTAL,"M",FALSE,0) )
				OpenTrolleyStep = 22;
			break;
		}
		case 22:
		{
/*Wait til Position is reached */
			if( isPositionOk(PAPERREMOVE_HORIZONTAL,PaperRemoveParameter.HorizontalPositions.TrolleyOpenRightStop,20) )
				OpenTrolleyStep = 24;

			break;
		}
		case 24:
		{
/*  move up */
			if( PapRemVerticalCmd(BOTH,CMD_SPEED,TRUE,PaperRemoveParameter.TrolleyOpenUpSpeed) )
			{
				OpenTrolleyStep = 25;
			}
			break;
		}
		case 25:
		{
/*  move up */
			if( PapRemVerticalCmd(BOTH,CMD_ABSOLUTE_POS,TRUE,PaperRemoveParameter.VerticalPositions.Up) )
			{
				OpenTrolleyStep = 26;
			}
			break;
		}
		case 26:
		{
/* Bewegung starten */
			if( PapRemVerticalCmd(BOTH,CMD_START_MOTION,FALSE,0L) )
			{
				OpenTrolleyStep = 27;
			}
			break;
		}
		case 27:
		{
/*Wait for UP*/
			if( isPapRemVerticalOk(BOTH,PaperRemoveParameter.VerticalPositions.Up,20) )
			{
				if( (GlobalParameter.TrolleyLeft != 0) && (GlobalParameter.TrolleyRight != 0) && OpenCounter ==1)
				{
					OpenCounter=2;
					OpenTrolleyStep = 10;
				}
				else
				OpenTrolleyStep = 29;
			}
			break;
		}
		case 29:
		{
/*set speed */
			if( SendMotorCmd(PAPERREMOVE_HORIZONTAL,"SP",1,PaperRemoveParameter.PaperRemoveSpeed) )
				OpenTrolleyStep = 30;
			break;
		}
		case 30:
		{
/*Paperremove is the next to do, so dont move back*/
			if (!PaperRemoveReady && GlobalParameter.PaperRemoveEnabled && START)
			{
				OpenTrolleyStep = 0;
				OpenTrolleyStart = 0;
				if( !DetectionError )
					TrolleyOpen = 1;
				break;
			}
/*Move Paper remove horizontically to wait pos*/
			if( SendMotorCmd(PAPERREMOVE_HORIZONTAL,"LA",1,PaperRemoveParameter.HorizontalPositions.EnableFeeder) )
				OpenTrolleyStep = 31;
			break;
		}
		case 31:
		{
/* Bewegung starten */
			if( SendMotorCmd(PAPERREMOVE_HORIZONTAL,"M",0,0) )
				OpenTrolleyStep = 32;
			break;
		}
		case 32:
		{
/*Wait til Position is reached */
			if( isPositionOk(PAPERREMOVE_HORIZONTAL,PaperRemoveParameter.HorizontalPositions.EnableFeeder,20) )
			{
				PaperRemoveReady = 0;
				OpenTrolleyStep = 0;
				OpenTrolleyStart = 0;
				if( !DetectionError )
					TrolleyOpen = 1;
			}
			break;
		}

/*****************************************/
/* special steps for trolley detection */
/*****************************************/
		case 50:
		{
			int i;
			CheckForPalette = FALSE;
			if(GlobalParameter.EnablePaletteLoading)
			{
				for(i=0;i<MAXTROLLEYS && !CheckForPalette;i++)
					if(Trolleys[i].NoCover)
						CheckForPalette = TRUE;
			}
			OpenTrolleyStep = 51;
			if(DetectCounter == 0)
			{
				StartPos = PaperRemoveParameter.TrolleyDetectStartPos;
				EndPos = PaperRemoveParameter.TrolleyDetectEndPos;
			}
			else
			{
				StartPos = abs(PaperRemoveParameter.TrolleyDetectStartPos) + GlobalParameter.TrolleyRightOffset;
				EndPos = abs(PaperRemoveParameter.TrolleyDetectEndPos) + GlobalParameter.TrolleyRightOffset;
			}
			/*
			 * safety check: Endpos must always be smaller than maximum position of Motor
			 */
			if( abs(EndPos) > abs(PAPERREMOVEHORIZONTAL_MAXPOS) )
				EndPos = PAPERREMOVEHORIZONTAL_MAXPOS;
			break;
		}
		case 51:
		{
/*Move Paper remove horizontically to trolley detect pos*/
			if( SendMotorCmd(PAPERREMOVE_HORIZONTAL,"LA",1,StartPos) )
				OpenTrolleyStep = 52;
			break;
		}

		case 52:
		{
/*set speed FAST*/
			if( SendMotorCmd(PAPERREMOVE_HORIZONTAL,"SP",1,PaperRemoveParameter.PaperRemoveSpeed) )
				OpenTrolleyStep = 55;
			break;
		}

		case 55:
		{
/* Bewegung starten */
			if( SendMotorCmd(PAPERREMOVE_HORIZONTAL,"M",0,0) )
				OpenTrolleyStep = 60;
			break;
		}
		case 60:
		{
/*Wait til Position is reached */
			if( !isPositionOk(PAPERREMOVE_HORIZONTAL,StartPos,20) )
				break;

			if(TrolleyCodeSensor)
			{
				OpenTrolleyStep = 65;
				DetectionError = 0;
			}
			else
			{
		/* FEHLER: kein Wagen */
				if(DetectCounter == 0)
				{
/*Wagen 1 (links) nicht gefunden: rechts probieren*/
					DetectCounter = 1;
					OpenTrolleyStep = 50;
					GlobalParameter.TrolleyLeft = 0;
				}
				else
				{
/*Wagen 2 (rechts) nicht gefunden*/
					DetectCounter = 0;
					GlobalParameter.TrolleyRight = 0;
/*no trolley found!*/
					if(GlobalParameter.TrolleyLeft == 0)
					{
/* check for palette*/
						if(CheckForPalette)
							OpenTrolleyStep = 150;
						else
						{
							AlarmBitField[13] = 1;
							DetectionError = 1;
							OrgBild = wBildAktuell;
							wBildNeu = 41;
							IgnoreButtons = 1;
							AbfrageOK = 0;
							OK_ButtonInv = 0;
							OK_CancelButtonInv = 1;
							AbfrageCancel = 0;
							AbfrageText1 = 5;
							AbfrageText2 = 0;
							AbfrageText3 = 7;
							AbfrageIcon = CAUTION;
							OpenTrolleyStep = 29;
						}
					}
					else
					{
/*nur Wagen links vorhanden: weiter mit Öffnen*/
						OpenTrolleyStep = 85;
					}
				}
			}
			break;
		}

		case 65:
		{
/*set speed */
			if( SendMotorCmd(PAPERREMOVE_HORIZONTAL,"SP",1,PaperRemoveParameter.TrolleyDetectSpeed) )
				OpenTrolleyStep = 70;
			break;
		}
		case 70:
		{
/*Move Paper remove horizontically to trolley detect end pos*/
			if( SendMotorCmd(PAPERREMOVE_HORIZONTAL,"LA",1,EndPos) )
				OpenTrolleyStep = 75;
			break;
		}

		case 75:
		{
/* Bewegung starten */
			if( SendMotorCmd(PAPERREMOVE_HORIZONTAL,"M",0,0) )
			{
				OpenTrolleyStep = 80;
				TrolleyCodeCounter.RESET = 1;
			}
			break;
		}
/* detect the edges of trolley sensor and wait til pos reached*/
		case 80:
		{
			TrolleyCodeCounter.RESET = 0;
			TrolleyCodeCounter.CU = !TrolleyCodeSensor;
			DetectedTrolley = TrolleyCodeCounter.CV;

/*Wait til Position is reached */
			if( isPositionOk(PAPERREMOVE_HORIZONTAL,EndPos,20) )
				OpenTrolleyStep = 84;

/*
 * longer than 3 sec no motion: error
 */
			OpenTrolleyTimer.IN = !Motors[PAPERREMOVE_HORIZONTAL].Moving;
			OpenTrolleyTimer.PT = 300; /* 3 sec */
			if( OpenTrolleyTimer.Q )
			{
				OpenTrolleyTimer.IN = 0;
				DetectionError = 1;
				OpenTrolleyStep = 29;
				AlarmBitField[14] = 1;
				OrgBild = wBildAktuell;
				wBildNeu = 41;
				IgnoreButtons = 1;
				AbfrageOK = 0;
				OK_ButtonInv = 0;
				OK_CancelButtonInv = 1;
				AbfrageCancel = 0;
				AbfrageText1 = 76;
				AbfrageText2 = 0;
				AbfrageText3 = 7;
				AbfrageIcon = CAUTION;
				GlobalParameter.TrolleyLeft = 0;
				GlobalParameter.TrolleyRight = 0;
			}
			break;
		}
		case 84:
		{
			DetectedTrolley = TrolleyCodeCounter.CV;
			TrolleyCodeCounter.RESET = 1;
	/* validate the code */
			if(DetectedTrolley>MAXTROLLEYS || DetectedTrolley<1)
			{
		/* FEHLER: ungültiger Code */

				DetectionError = 1;
				OpenTrolleyStep = 29;
				AlarmBitField[14] = 1;
				OrgBild = wBildAktuell;
				wBildNeu = 41;
				IgnoreButtons = 1;
				AbfrageOK = 0;
				OK_ButtonInv = 0;
				OK_CancelButtonInv = 1;
				AbfrageCancel = 0;
				AbfrageText1 = 6;
				AbfrageText2 = 0;
				AbfrageText3 = 7;
				AbfrageIcon = CAUTION;
				GlobalParameter.TrolleyLeft = 0;
				GlobalParameter.TrolleyRight = 0;
			}
			else
			{
		/*code eintragen*/
				if(PaletteDetection)
				{
/* plausibility: Palette code found, but not marked as palette ->Error*/
					if(Trolleys[DetectedTrolley].NoCover)
						GlobalParameter.TrolleyLeft = DetectedTrolley;
					else
					{
				/* ERROR: invalid Code */
						ShowMessage(6,81,7, CAUTION, OKONLY, TRUE);
						DetectionError = TRUE;
						AlarmBitField[14] = TRUE;
						GlobalParameter.TrolleyLeft = NO_TROLLEY;
						GlobalParameter.TrolleyRight = NO_TROLLEY;
						PaletteDetection = FALSE;
						OpenTrolleyStep = 29;
						OpenTrolleyTimer.IN = FALSE;
						break;
					}

					PaletteDetection = FALSE;
					OpenTrolleyStep = 85;
					OpenTrolleyTimer.IN = FALSE;
				}
				else
				if(DetectCounter == 0) /*1st detection: left trolley*/
				{
					GlobalParameter.TrolleyLeft = DetectedTrolley;
/* plausibility: Palette code found during trolley detection ->Error*/
					if(Trolleys[DetectedTrolley].NoCover)
					{
				/* ERROR: invalid Code */
						ShowMessage(6,80,7, CAUTION, OKONLY, TRUE);
						DetectionError = TRUE;
						AlarmBitField[14] = TRUE;
						GlobalParameter.TrolleyLeft = NO_TROLLEY;
						GlobalParameter.TrolleyRight = NO_TROLLEY;
						PaletteDetection = FALSE;
						OpenTrolleyStep = 29;
						OpenTrolleyTimer.IN = FALSE;
						break;
					}

					if(Trolleys[GlobalParameter.TrolleyLeft].Double)
					{
						GlobalParameter.TrolleyRight = 0;
			/*READY, no second detection required*/
						DetectCounter = 0;
						OpenTrolleyStep = 85;
						break;
					}
					else
					{
						DetectCounter = 1;
						OpenTrolleyStep = 50;
						break;
					}
				}
				else  /*2nd detection: right trolley*/
				{
					GlobalParameter.TrolleyRight = DetectedTrolley;
		/*validation*/
					if(Trolleys[GlobalParameter.TrolleyRight].Double)
					{
						DetectionError = 1;
						OpenTrolleyStep = 29;
						DetectCounter = 0;
						GlobalParameter.TrolleyRight = 0;
						GlobalParameter.TrolleyLeft = 0;
						AlarmBitField[14] = 1;
						OrgBild = wBildAktuell;
						wBildNeu = 41;
						OK_ButtonInv = 0;
						OK_CancelButtonInv = 1;
						IgnoreButtons = 1;
						AbfrageOK = 0;
						AbfrageCancel = 0;
						AbfrageText1 = 6;
						AbfrageText2 = 93;
						AbfrageText3 = 7;
						AbfrageIcon = CAUTION;
					}
					else
					{
						DetectCounter = 0;
						OpenTrolleyStep = 85;
					}
				}
			}
			break;
		}

		case 85:
		{
			TrolleyCodeCounter.RESET = 0;

/*reset speed to fast*/
			if( SendMotorCmd(PAPERREMOVE_HORIZONTAL,"SP",1,PaperRemoveParameter.PaperRemoveSpeed) )
				OpenTrolleyStep = 90;
			break;
		}

		case 90:
		{
			OpenTrolleyStep = 8;
			break;
		}

/**************************************************************************/
/**************************************************************************/
/**************************************************************************/
		case 150:
		{
			PaletteDetection = TRUE;
			StartPos = labs(PaperRemoveParameter.HorizontalPositions.PaletteDetectStartPos);
			EndPos = labs(PaperRemoveParameter.HorizontalPositions.PaletteDetectEndPos);
			/*
			 * safety check: Endpos must always be smaller than maximum position of Motor
			 */
			if( labs(EndPos) > labs(PAPERREMOVEHORIZONTAL_MAXPOS) )
				EndPos = PAPERREMOVEHORIZONTAL_MAXPOS;

			OpenTrolleyStep = 151;
			OpenTrolleyTimer.IN = FALSE;
			break;
		}
		case 151:
		{
/*Move Paper remove horizontally to Palette detect pos*/
			if( SendMotorCmd(PAPERREMOVE_HORIZONTAL,"LA",1,StartPos) )
			{
				OpenTrolleyStep = 152;
				OpenTrolleyTimer.IN = FALSE;
				break;
			}
			break;
		}
		case 152:
		{
/*set speed FAST*/
			if( SendMotorCmd(PAPERREMOVE_HORIZONTAL,"SP",1,PaperRemoveParameter.PaperRemoveSpeed) )
			{
				OpenTrolleyStep = 155;
				OpenTrolleyTimer.IN = FALSE;
				break;
			}
			break;
		}
		case 155:
		{
/* Bewegung starten */
			if( SendMotorCmd(PAPERREMOVE_HORIZONTAL,"M",0,0) )
			{
				OpenTrolleyStep = 160;
				OpenTrolleyTimer.IN = FALSE;
				break;
			}
			break;
		}

		case 160:
		{
/*Wait til Position is reached */
			if( isPositionOk(PAPERREMOVE_HORIZONTAL,StartPos,20) )
			{
			{
				OpenTrolleyStep = 161;
				OpenTrolleyTimer.IN = FALSE;
				break;
			}
				break;
			}
			break;
		}

		case 161:
		{
/*Move Paper remove horizontally to Palette detect pos*/
			if( SendMotorCmd(PAPERREMOVE_HORIZONTAL,"LA",1,EndPos) )
			{
				OpenTrolleyStep = 162;
				OpenTrolleyTimer.IN = FALSE;
				break;
			}
			break;
		}
		case 162:
		{
/*set speed FAST*/
			if( SendMotorCmd(PAPERREMOVE_HORIZONTAL,"SP",1,PaperRemoveParameter.PaletteDetectSpeed) )
			{
				OpenTrolleyStep = 165;
				OpenTrolleyTimer.IN = FALSE;
				break;
			}
			break;
		}
		case 165:
		{
/* Bewegung starten */
			TrolleyCodeCounter.RESET = 1;
			if( SendMotorCmd(PAPERREMOVE_HORIZONTAL,"M",0,0) )
			{
				OpenTrolleyStep = 170;
				OpenTrolleyTimer.IN = FALSE;
				break;
			}
			break;
		}

/* detect the edges of trolley sensor and wait til pos reached*/
		case 170:
		{
			TrolleyCodeCounter.RESET = 0;
			TrolleyCodeCounter.CU = TrolleyCodeSensor;

/*Wait til Position is reached */
			if( isPositionOk(PAPERREMOVE_HORIZONTAL,EndPos,20) )
			{
				OpenTrolleyStep = 84;
				OpenTrolleyTimer.IN = FALSE;
				break;
			}
			break;
		}

	}/*switch*/

	CTU(&TrolleyCodeCounter);

}
```

#### closetrolley.c
```c
#ifdef _DEFAULT_INCLUDES
	#include <AsDefault.h>
#endif
/****************************************************************************/
/*	Ablauf Plattenwagen schliessen */
/*																			*/
/*																			*/
/*	Versionsgeschichte:														*/
/*  Version		Datum		Änderung								von		*/
/*	1.00		10.09.02	erste Implementation					HA		*/
/*	1.10		16.09.02	Trolley offen/geschlossen jetzt mit		HA		*/
/*							2 Positionen (start und ende der Bewegung		*/
/*	1.20		02.01.03	vor oeffnen/schließen wird jetzt der	HA		*/
/*							Vertikalantrieb Referenz gefahren				*/
/*	1.30		06.01.03	Verschluß "nachdruecken" rausgenommen	HA		*/
/*							(neuer Verschluß -> nicht mehr nötig)			*/
/*																			*/
/*																			*/
/****************************************************************************/

#include "glob_var.h"
#include "in_out.h"
#include "asstring.h"
#include <string.h>
#include "motorfunc.h"
#include "auxfunc.h"

#define PRELIFT	300
#define PUSHPOS_H 3157
#define PUSHPOS_V 400
#define BACKWAY_AFTER_CLOSING (100) /* relativ in Incr. */

_LOCAL	USINT	CloseTrolleyStep;
_GLOBAL	BOOL	CloseTrolleyStart;
_LOCAL TON_10ms_typ CloseTrolleyTimer;
USINT			tmp[20];

_GLOBAL	BOOL	CloseTrolleyReady;
_GLOBAL	BOOL	OpenTrolleyStart;
_GLOBAL 	BOOL	CloseTrolleyTriggeredCloseDrawer;

USINT	CloseCounter; /* for max 2 cycles (2 single trolleys)*/
BOOL Small;

void CloseTrolley(void)
{
	/* Motoren keine Referenz? -> Ende*/
	if( !Motors[PAPERREMOVE_VERTICAL].ReferenceOk
	||  !Motors[PAPERREMOVE_VERTICAL2].ReferenceOk
	)
		 return;

	if( !Motors[PAPERREMOVE_HORIZONTAL].ReferenceOk ) return;
	if( !Motors[FEEDER_VERTICAL].ReferenceOk ) return;

	TON_10ms(&CloseTrolleyTimer);

	if (!CloseTrolleyStart)
	{
		CloseTrolleyStep=0;
		CloseTrolleyTriggeredCloseDrawer = 0;
	}

	switch (CloseTrolleyStep)
	{
		case 0:
		{
/* wait for start command */
			if (!CloseTrolleyStart || PaperRemoveStart || OpenTrolleyStart) break;
/*enable conditions*/

/*check, if Feeder is out of collision area (should be the case here)*/
			if( abs(Motors[FEEDER_VERTICAL].Position) > abs(FeederParameter.VerticalPositions.EnablePaperRemove)+20 )
				break;

/*NEW*/
			CloseCounter = 1;

/*NEW always do a reference of paperremove vert. at first */
			CloseTrolleyStep = 4;
			break;
		}

		case 1:
		{
/* else move up */
			if( PapRemVerticalCmd(BOTH,CMD_ABSOLUTE_POS,TRUE,PaperRemoveParameter.VerticalPositions.Up) )
			{
				CloseTrolleyStep = 2;
			}
			break;
		}
		case 2:
		{
/* Bewegung starten */
			if( PapRemVerticalCmd(BOTH,CMD_START_MOTION,FALSE,0L) )
			{
				CloseTrolleyStep = 3;
			}
			break;
		}
		case 3:
		{
/*Wait for UP*/
			if( isPapRemVerticalOk(BOTH,PaperRemoveParameter.VerticalPositions.Up,20) )
				CloseTrolleyStep = 8;
			break;
		}

/*NEW paperremove vert reference at first*/
		case 4:
		{
			Motors[PAPERREMOVE_VERTICAL].StartRef = 1;
			Motors[PAPERREMOVE_VERTICAL].ReferenceOk = 0;
			Motors[PAPERREMOVE_VERTICAL2].StartRef = 1;
			Motors[PAPERREMOVE_VERTICAL2].ReferenceOk = 0;
			CloseTrolleyStep = 5;
			break;
		}
		case 5:
		{
			if( Motors[PAPERREMOVE_VERTICAL].ReferenceOk == 0
			 || Motors[PAPERREMOVE_VERTICAL2].ReferenceOk == 0
			)
				break;

			CloseTrolleyStep = 8;

			break;
		}

		case 8:
		{
			if(  (Out_PaperGripOn[LEFT] == OFF)
			  && (Out_PaperGripOn[RIGHT] == OFF)
			  && CloseTrolleyTimer.Q )
			{
				CloseTrolleyStep = 10;
				CloseTrolleyTimer.IN = 0;
				break;
			}

			Out_PaperGripOn[LEFT] = OFF;
			Out_PaperGripOn[RIGHT] = OFF;
			CloseTrolleyTimer.IN = TRUE;
			CloseTrolleyTimer.PT = PaperRemoveParameter.GripOffTime;
			break;
		}

/*********************************************************/
/*move fast to "trolley open" pos*/
/*********************************************************/
		case 10:
		{
/*NEW*/
			if( (GlobalParameter.TrolleyLeft != 0) && CloseCounter == 1)
			{
				if(GlobalParameter.EnablePaletteLoading && Trolleys[GlobalParameter.TrolleyLeft].NoCover)
				{
					CloseTrolleyStart = FALSE;
					TrolleyOpen = FALSE;
					CloseTrolleyStep = 0;
					CloseTrolleyTimer.IN = 0;
					break;
				}

				PaperRemoveParameter.HorizontalPositions.TrolleyOpenRightStart = Trolleys[GlobalParameter.TrolleyLeft].OpenStart;
				PaperRemoveParameter.HorizontalPositions.TrolleyOpenRightStop = Trolleys[GlobalParameter.TrolleyLeft].OpenStop;
				PaperRemoveParameter.HorizontalPositions.TrolleyCloseRightStart = Trolleys[GlobalParameter.TrolleyLeft].CloseStart;
				PaperRemoveParameter.HorizontalPositions.TrolleyCloseRightStop = Trolleys[GlobalParameter.TrolleyLeft].CloseStop;
				if(Trolleys[GlobalParameter.TrolleyLeft].Double)
					Small = 0;
				else
					Small = 1;
			}
			if( (GlobalParameter.TrolleyRight != 0 && CloseCounter == 2)
			||  (GlobalParameter.TrolleyLeft == 0 && GlobalParameter.TrolleyRight != 0 && CloseCounter == 1 ) )
			{
				PaperRemoveParameter.HorizontalPositions.TrolleyOpenRightStart = abs(Trolleys[GlobalParameter.TrolleyRight].OpenStart) + GlobalParameter.TrolleyRightOffset;
				PaperRemoveParameter.HorizontalPositions.TrolleyOpenRightStop = abs(Trolleys[GlobalParameter.TrolleyRight].OpenStop) + GlobalParameter.TrolleyRightOffset;
				PaperRemoveParameter.HorizontalPositions.TrolleyCloseRightStart = abs(Trolleys[GlobalParameter.TrolleyRight].CloseStart) + GlobalParameter.TrolleyRightOffset;
				PaperRemoveParameter.HorizontalPositions.TrolleyCloseRightStop = abs(Trolleys[GlobalParameter.TrolleyRight].CloseStop) + GlobalParameter.TrolleyRightOffset;
				Small = 1;
			}

/*check, if Feeder is out of collision area (should be the case here)*/
			if( abs(Motors[FEEDER_VERTICAL].Position) > abs(FeederParameter.VerticalPositions.EnablePaperRemove)+20 )
				break;

/*Move Paper remove horizontically to open trolley pos*/
			if( SendMotorCmd(PAPERREMOVE_HORIZONTAL,"LA",1,PaperRemoveParameter.HorizontalPositions.TrolleyCloseRightStart) )
				CloseTrolleyStep = 11;
			break;
		}
		case 11:
		{
/* Bewegung starten */
			if( SendMotorCmd(PAPERREMOVE_HORIZONTAL,"M",0,0) )
				CloseTrolleyStep = 12;
			break;
		}
		case 12:
		{
/*Wait til Position is reached */
			if( isPositionOk(PAPERREMOVE_HORIZONTAL,PaperRemoveParameter.HorizontalPositions.TrolleyCloseRightStart,20) )
				CloseTrolleyStep = 14;

			break;
		}

/*********************************************************/
/*move down slowly on trolley */
/*********************************************************/
		case 14:
		{
/* Paper remove down on trolley*/
			if( PapRemVerticalCmd(BOTH,CMD_SPEED,TRUE,PaperRemoveParameter.TrolleyOpenDownSpeed) )
			{
				CloseTrolleyStep = 15;
			}
			break;
		}
		case 15:
		{
/* Paper remove down on trolley*/
			if( PapRemVerticalCmd(BOTH,CMD_ABSOLUTE_POS,TRUE,PaperRemoveParameter.VerticalPositions.OnTrolley) )
			{
				CloseTrolleyStep = 16;
			}
			break;
		}
		case 16:
		{
/* Bewegung starten */
			if( PapRemVerticalCmd(BOTH,CMD_START_MOTION,FALSE,0L) )
			{
				CloseTrolleyStep = 17;
			}
			break;
		}
		case 17:
		{
/*Wait for pos on trolley*/
			if( isPapRemVerticalOk(BOTH,PaperRemoveParameter.VerticalPositions.OnTrolley,20)
			|| ( CloseTrolleyTimer.Q ))
			{
				CloseTrolleyStep = 19;
				CloseTrolleyTimer.IN = 0;
				break;
			}

			CloseTrolleyTimer.IN = 1;
			CloseTrolleyTimer.PT = PaperRemoveParameter.TimeoutOnTrolley;
			break;
		}

/*********************************************************/
/*move slowly to "trolley closed" pos */
/*********************************************************/
		case 19:
		{
/*Move Paper remove horizontically to closed trolley pos*/
			if( SendMotorCmd(PAPERREMOVE_HORIZONTAL,"LA",1,PaperRemoveParameter.HorizontalPositions.TrolleyCloseRightStop) )
				CloseTrolleyStep = 20;
			break;
		}
		case 20:
		{
/*set speed */
			if( SendMotorCmd(PAPERREMOVE_HORIZONTAL,"SP",1,PaperRemoveParameter.TrolleyOpenCloseSpeed) )
				CloseTrolleyStep = 21;
			break;
		}
		case 21:
		{
/* Bewegung starten */
			if( SendMotorCmd(PAPERREMOVE_HORIZONTAL,"M",0,0) )
				CloseTrolleyStep = 22;
			break;
		}
		case 22:
		{
/*Wait til Position is reached */
			if( isPositionOk(PAPERREMOVE_HORIZONTAL,PaperRemoveParameter.HorizontalPositions.TrolleyCloseRightStop,20)
			|| ( CloseTrolleyTimer.Q ))
			{
				CloseTrolleyStep = 28;
				CloseTrolleyTimer.IN = 0;
				break;
			}

			CloseTrolleyTimer.IN = 1;
			if(Small)
				CloseTrolleyTimer.PT = PaperRemoveParameter.TimeoutOpenTrolleySmall;
			else
				CloseTrolleyTimer.PT = PaperRemoveParameter.TimeoutOpenTrolleyBig;
			break;

		}

/*HA 05.05.03 V1.05 steps 28-30*/
/*********************************************************/
/*move back a little to release shutter */
/*********************************************************/
		case 28:
		{
/*Move Paper remove horizontically back a little (to open start position actually)*/
			if( SendMotorCmd(PAPERREMOVE_HORIZONTAL,"LA",1,PaperRemoveParameter.HorizontalPositions.TrolleyCloseRightStop+BACKWAY_AFTER_CLOSING) )
				CloseTrolleyStep = 29;
			break;
		}
		case 29:
		{
/* Bewegung starten */
			if( SendMotorCmd(PAPERREMOVE_HORIZONTAL,"M",0,0) )
				CloseTrolleyStep = 30;
			break;
		}
		case 30:
		{
/*Wait til Position is reached */
			if( isPositionOk(PAPERREMOVE_HORIZONTAL,PaperRemoveParameter.HorizontalPositions.TrolleyCloseRightStop+BACKWAY_AFTER_CLOSING,20) )
				CloseTrolleyStep = 44;
			break;
		}

/*********************************************************/
/*move up fast completely */
/*********************************************************/
		case 44:
		{
/*  move up */
			if( PapRemVerticalCmd(BOTH,CMD_SPEED,TRUE,PaperRemoveParameter.TrolleyOpenUpSpeed) )
			{
				CloseTrolleyStep = 45;
			}
			break;
		}
		case 45:
		{
/*  move up */
			if( PapRemVerticalCmd(BOTH,CMD_ABSOLUTE_POS,TRUE,PaperRemoveParameter.VerticalPositions.Up) )
			{
				CloseTrolleyStep = 46;
			}
			break;
		}
		case 46:
		{
/* Bewegung starten */
			if( PapRemVerticalCmd(BOTH,CMD_START_MOTION,FALSE,0L) )
			{
				CloseTrolleyStep = 47;
			}
			break;
		}
		case 47:
		{
/*Wait for UP*/
			if( isPapRemVerticalOk(BOTH,PaperRemoveParameter.VerticalPositions.Up,20)
			|| ( CloseTrolleyTimer.Q ))
			{

/* HA 24.04.03 V1.05 bugfix: closing 2nd trolley was not activated (if-construct was missing)*/
				if( (GlobalParameter.TrolleyLeft != 0) && (GlobalParameter.TrolleyRight != 0) && CloseCounter ==1)
				{
					CloseCounter = 2;
					CloseTrolleyStep = 10;
				}
				else
					CloseTrolleyStep = 79;
				CloseTrolleyTimer.IN = 0;
				break;
			}
			CloseTrolleyTimer.IN = 1;
			CloseTrolleyTimer.PT = PaperRemoveParameter.TimeoutUpFromTrolley;
			break;

		}

/*********************************************************/
/*move back fast to wait pos*/
/*********************************************************/

		case 79:
		{
/*set speed */
			if( SendMotorCmd(PAPERREMOVE_HORIZONTAL,"SP",1,PaperRemoveParameter.PaperRemoveSpeed) )
				CloseTrolleyStep = 80;
			break;
		}
		case 80:
		{
/*Move Paper remove horizontically to wait pos*/
			if( SendMotorCmd(PAPERREMOVE_HORIZONTAL,"LA",1,PaperRemoveParameter.HorizontalPositions.EnableFeeder) )
				CloseTrolleyStep = 81;
			break;
		}
		case 81:
		{
/* Bewegung starten */
			if( SendMotorCmd(PAPERREMOVE_HORIZONTAL,"M",0,0) )
				CloseTrolleyStep = 82;
			break;
		}
		case 82:
		{
/*Wait til Position is reached */
			if( isPositionOk(PAPERREMOVE_HORIZONTAL,PaperRemoveParameter.HorizontalPositions.EnableFeeder,20) )
			{
				CloseTrolleyStep = 0;
				CloseTrolleyStart = 0;
				TrolleyOpen = 0;
			}
			break;
		}
	}/*switch*/
}
```

- motorfunc.h (reference to Logical/GlobalIncludes/motorfunc.h)

#### motorfunc.c
```c
#ifdef _DEFAULT_INCLUDES
	#include <AsDefault.h>
#endif
/*
                             *******************
******************************* C SOURCE FILE *******************************
**                           *******************                           **
**                                                                         **
** project  : LS JET II                                                    **
** filename : MOTORFUNC.C                                                  **
** version  : 1.02                                                         **
** date     : 07.11.2007                                                   **
**                                                                         **
*****************************************************************************
** Abstract                                                                **
** ========                                                                **
** Implementation of motor control functions (sending commands and         **
** check for positions)                                                    **
**                                                                         **
** Copyright (c) 2007, Krause-Biagosch GmbH                                **
** All rights reserved.                                                    **
**                                                                         **
*****************************************************************************
VERSION HISTORY:
----------------
Version     : 1.00
Date        : 20.10.2006
Revised by  : Herbert Aden
Description : Original version.

Version     : 1.01
Date        : 12.10.2007
Revised by  : Herbert Aden
Description : - a variable for holding the current step in function MoveToAbsPosition
                must now be provided by the caller (a pointer to that var of course!)
              - in Fct. IsPositionOK the check for being in a certain position window
                failed, if that window was 0, i.e. if an exact position is to be found
                the expression "currpos - checkpos < deviation" results in false, so it
                was changed to "currpos - checkpos <= deviation" so that if
                currpos==checkpos the result is still true for deviaition==0

Version     : 1.02
Date        : 07.11.2007
Revised by  : Herbert Aden
Description : - bugfix: in RequestMotorData the var SerialCmd.Request was set TRUE
                unconditionally. Caused sporadic Errormessages for serial comm.

*/
#define _MOTORFUNC_C_SRC

/****************************************************************************/
/**                                                                        **/
/**                           INCLUDE FILES                                **/
/**                                                                        **/
/****************************************************************************/
#include <stdlib.h>
#include <string.h>
#include "glob_var.h"

#include "motorfunc.h"

/****************************************************************************/
/**                                                                        **/
/**                       DEFINITIONS AND MACROS                           **/
/**                                                                        **/
/****************************************************************************/
/* NONE */

/****************************************************************************/
/**                                                                        **/
/**                      EXPORTED VARIABLES                                **/
/**                                                                        **/
/****************************************************************************/
/*@checked@*/
_GLOBAL   SerialCmd_Typ       SerialCmd;

/****************************************************************************/
/**                                                                        **/
/**                           GLOBAL VARIABLES                             **/
/**                                                                        **/
/****************************************************************************/
static  BOOL                  Send1Ready = 0;

/****************************************************************************/
/**                                                                        **/
/**                          EXPORTED FUNCTIONS                            **/
/**                                                                        **/
/****************************************************************************/

/****************************************************************************/
/** Send commands to a motor                                                */
/****************************************************************************/
BOOL	SendMotorCmd(const INT pMotor,const char *CmdStr,const BOOL UseValue,const DINT Value)
{
	if(SerialCmd.Send == FALSE) /*wait, till no other sending active*/
	{
		strcpy(SerialCmd.CmdString,CmdStr);
		SerialCmd.UseParameter = UseValue;
		SerialCmd.Parameter = Value;
		if (   (STREQ(CmdStr,CMD_ABSOLUTE_POS))
			|| (STREQ(CmdStr,CMD_RELATIVE_POS))
			|| (STREQ(CmdStr,CMD_MOVE_AT))
		  ) /*bei LA oder LR oder V Refdir verwenden, sonst nicht*/
			SerialCmd.UseRefDirection = TRUE;
		else
			SerialCmd.UseRefDirection = FALSE;

		SerialCmd.SendMotor = pMotor;
		SerialCmd.Send = TRUE;
		return TRUE;
	}
	else
		return FALSE;
}

/****************************************************************************/
/** Request data from a motor                                                */
/****************************************************************************/
BOOL	RequestMotorData(const INT pMotor,const char *CmdString)
{
	if( SerialCmd.Send == TRUE )
		return FALSE;
	else
	{
		SerialCmd.Request = TRUE;
		return SendMotorCmd(pMotor,CmdString,FALSE,0);
	}
}

/****************************************************************************/
/** Check, if a motor is in a certain position window                       */
/****************************************************************************/
BOOL	isPositionOk(const INT Motor,const DINT Pos,const DINT Deviation)
{
	DINT tmp;
	if (labs(Deviation) > 0 )
		tmp = labs(Deviation);
	else	/* if Dev is 0, then use deviation defined in motorparam*/
		tmp = labs(Motors[Motor].Parameter.PositionWindow);

	if( labs( labs(Motors[Motor].Position) - labs(Pos) ) <= tmp )
		return TRUE;
	else
		return FALSE;
}

/****************************************************************************/
/** Check, if a motor is below a certain position                           */
/****************************************************************************/
BOOL	isPositionLowerThan(const INT Motor,DINT Pos)
{
	if( labs(Motors[Motor].Position) < (labs(Pos) ) )
		return TRUE;
	else
		return FALSE;
}

/****************************************************************************/
/** Check, if a motor is above a certain position                           */
/****************************************************************************/
BOOL	isPositionHigherThan(const INT Motor,DINT Pos)
{
	if( labs(Motors[Motor].Position) > (labs(Pos) ) )
		return TRUE;
	else
		return FALSE;
}

/****************************************************************************/
/* send commands to paper remove vertical */
/****************************************************************************/
BOOL	PapRemVerticalCmd(BOOL Config,char *CmdString,BOOL UseValue,DINT Value)
{
	if(Config == LEFT)
		return SendMotorCmd(PAPERREMOVE_VERTICAL, CmdString, UseValue, Value);
	else
	if(Config == RIGHT)
		return SendMotorCmd(PAPERREMOVE_VERTICAL2, CmdString, UseValue, Value);
	else
	if ( Send1Ready == FALSE )
	{
		if( SendMotorCmd(PAPERREMOVE_VERTICAL, CmdString, UseValue, Value) )
			Send1Ready = TRUE;

		return FALSE;
	}
	else
	{
		if( SendMotorCmd(PAPERREMOVE_VERTICAL2, CmdString, UseValue, Value) )
		{
			Send1Ready = FALSE;
			return TRUE;
		}
		return FALSE;
	}
}

/****************************************************************************/
/* Check position of paper remove vertical */
/****************************************************************************/
BOOL	isPapRemVerticalOk(BOOL Config,DINT Pos,UDINT MaxDeviation)
{
	if(Config == LEFT)
		return isPositionOk(PAPERREMOVE_VERTICAL, Pos, MaxDeviation);
	else
	if(Config == RIGHT)
		return isPositionOk(PAPERREMOVE_VERTICAL2, Pos, MaxDeviation);
	else
	if ( isPositionOk(PAPERREMOVE_VERTICAL, Pos, MaxDeviation) )
	{
		if ( isPositionOk(PAPERREMOVE_VERTICAL2, Pos, MaxDeviation) )
			return TRUE;
		else
			return FALSE;
	}
	else
		return FALSE;
}

/****************************************************************************/
/* move motor to an absolute position and wait for motion to start */
/****************************************************************************/
BOOL  MoveToAbsPosition(INT pMotor, DINT Pos, DINT Speed, USINT *pStep)
{
	int step = *pStep;

	BOOL retval = FALSE;

	if (pMotor == 0 && Pos == 0L && Speed == 0L)
	{
		step = 0;
		*pStep = 0;
		return FALSE;
	}

	switch (step)
	{
		case 0:
		{
/* send target position */
			if( SendMotorCmd(pMotor,CMD_ABSOLUTE_POS,TRUE,Pos) )
			{
				if ( Speed == DONT_SEND_SPEED )
					step = 20;
				else
					step = 10;
			}
			retval = FALSE;
			break;
		}
/* set speed */
		case 10:
		{
			if( SendMotorCmd(pMotor,CMD_SPEED,TRUE,Speed) )
			{
				step = 20;
			}
			retval = FALSE;
			break;
		}
		case 20:
		{
/* start motion */
			if( SendMotorCmd(pMotor,CMD_START_MOTION,FALSE,0L) )
			{
				step = 30;
			}
			retval = FALSE;
			break;
		}
		case 30:
		{
/* Wait til motion begins or Motor is in position (might be already there!)*/
			if( Motors[pMotor].Moving
			    ||
			    isPositionOk(pMotor,Pos,0) )
			{
				step = 0;
				retval = TRUE;
			}
			break;
		}
	}
	*pStep = step;
	return retval;
}

/****************************************************************************/
/* move motor to an relative position without waiting for motion to start */
/****************************************************************************/
BOOL  MoveToRelPosition(INT pMotor, DINT Pos, DINT Speed, USINT *pStep)
{
	int step = *pStep;

	BOOL retval = FALSE;

	if (pMotor == 0 && Pos == 0L && Speed == 0L)
	{
		step = 0;
		*pStep = 0;
		return FALSE;
	}

	switch (step)
	{
		case 0:
		{
/* send target position */
			if( SendMotorCmd(pMotor,CMD_RELATIVE_POS,TRUE,Pos) )
			{
				if ( Speed == DONT_SEND_SPEED )
					step = 20;
				else
					step = 10;
			}
			retval = FALSE;
			break;
		}
/* set speed */
		case 10:
		{
			if( SendMotorCmd(pMotor,CMD_SPEED,TRUE,Speed) )
			{
				step = 20;
			}
			retval = FALSE;
			break;
		}
		case 20:
		{
/* start motion */
			if( SendMotorCmd(pMotor,CMD_START_MOTION,FALSE,0L) )
			{
				step = 30;
			}
			retval = FALSE;
			break;
		}
		case 30:
		{
			step = 0;
			retval = TRUE;
			break;
		}
	}
	*pStep = step;
	return retval;
}

/****************************************************************************/
/**                                                                        **/
/**                          LOCAL FUNCTIONS                               **/
/**                                                                        **/
/****************************************************************************/
/* NONE */

/****************************************************************************/
/**                                                                        **/
/**                                 EOF                                    **/
/**                                                                        **/
/****************************************************************************/
```

- auxfunc.c (reference to Logical/Exposer/Ablauf/papentf/auxfunc.c)

- auxfunc.h (reference to Logical/GlobalIncludes/auxfunc.h)

### Program Logical/Exposer/Ablauf/referenz (ANSIC, version 1.01.0) - Gesamt Referenzfahrt
